// TIA Portal project "data_connection" (V17)

(* hardware
DEVICE "S7-1200 station_1"  S7-1200 Station
   slot 0: "Rack_0"  S7-1200 Rack  Rack  V1.0
   slot 1: "PLC_1"  CPU 1211C AC/DC/Rly  6ES7 211-1BE40-0XB0  V4.4
*)

// ===== PLC "PLC_1"  CPU 1211C AC/DC/Rly =====

DATA_BLOCK "data_connection_test"   // DB1
{ S7_Optimized_Access := 'TRUE' }
VERSION : 0.1
// stored: InstanceOfName DataConnectionTest
"DataConnectionTest"
BEGIN
END_DATA_BLOCK

FUNCTION_BLOCK "DataConnectionTest"   // FB1, SCL
{ S7_Optimized_Access := 'TRUE' }
VERSION : 0.1
   VAR
      opc_ua : Struct
         test_string : String;
         test_bool : Bool;
         test_real : Real;
         test_int : Int;
         test_wstring : WString;
      END_STRUCT;
   END_VAR
BEGIN
END_FUNCTION_BLOCK

ORGANIZATION_BLOCK "Main"   // OB1, LAD, ProgramCycle
TITLE = "Main Program Sweep (Cycle)"
{ S7_Optimized_Access := 'TRUE' }
VERSION : 0.1
   VAR_INPUT
      Initial_Call : Bool;   // Initial call of this OB
      Remanence : Bool;   // =True, if remanent data are available
   END_VAR
BEGIN

REGION Network 1
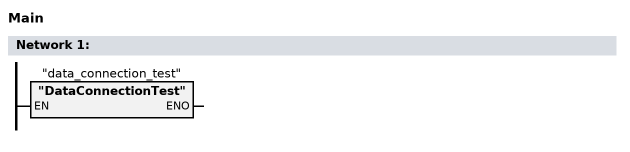
   RUNG wire#powerrail
      "data_connection_test"()
   END_RUNG
   // the same network as SCL:
   "data_connection_test"();   // "DataConnectionTest"
END_REGION
END_ORGANIZATION_BLOCK